ABB RobotStudio station: CubesMovement_20241125-112948.rsstn

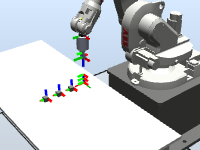
Station CubesMovement (saved by RobotStudio 6.8.8307.1040)
Controller System1, task T_ROB1: task frame (RAPID world) sits at (0, 0, 520) mm in the station
Controller System1
  mechanical unit ROB_1: IRB1600_10_145__01, 6 joints, base frame (0, 0, 0) mm
Layout (positions relative to the parent item):
  - IRB1600_10_145__01 [mechanism, from Robots\IRB1600_10_145_G_01.rslib] at (0, 0, 520) mm; joint values [-0.0068, 0.3691, 0.5943, 0, 0.6074, 1.564] (rad or m)
  - base [part, from Desktop\подставка.rslib]
  - table [part, from Desktop\Стол сборка.rslib] at (677.65, -723.32, 0) mm, rotated rx 0 ry 0 rz 90 deg
  - toolGripper [mechanism, from Desktop\toolGripper.rslib] at (744.98, -5.05, 1101.68) mm, rotated rx 180 ry 0 rz 90 deg
  - cube_1 [part, from Desktop\cube.rslib] at (844.98, -5.05, 730.16) mm
  - cube_2 [part, from Desktop\cube.rslib] at (944.98, -5.05, 730.39) mm
  - cube_3 [part, from Desktop\cube.rslib] at (1044.98, -5.05, 730.61) mm
Attachment: wobjTable is attached to table
Attachment: toolGripper is attached to IRB1600_10_145__01 / Link6
Collision set CollisionSet_1: IRB1600_10_145__01, toolGripper, table against table, toolGripper, near miss 0 m
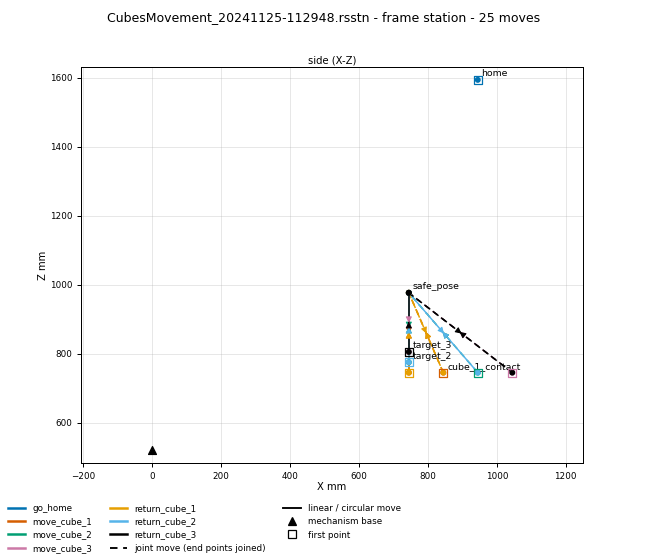
[picture p0: tool path of CubesMovement_20241125-112948.rsstn in frame station, 25 of 25 moves have a stored position in this frame; points joined in program order, loops and branches not executed]
Targets, tools, work objects and paths stored in the station, written as RAPID:
! task T_ROB1
MODULE CalibData
  PERS tooldata toolGripper:=[TRUE,[[0,0,160],[1,0,0,0]],[0.8,[0,0,1],[1,0,0,0],0,0,0]];
  TASK PERS wobjdata wobjTable:=[FALSE,TRUE,"",[[744.979,-5.048,210.071],[1,0,0,0]],[[0,0,0],[1,0,0,0]]];
ENDMODULE

! task T_ROB1
MODULE Module1
  CONST robtarget home:=[[944.855715851,0,1074],[0.5,0,0.866025404,0],[0,0,0,0],[9E+09,9E+09,9E+09,9E+09,9E+09,9E+09]];
  CONST robtarget cube_1_pose:=[[100,0,0],[1,0,0,0],[0,0,0,0],[9E+09,9E+09,9E+09,9E+09,9E+09,9E+09]];
  CONST robtarget cube_2_pose:=[[200,0,0],[1,0,0,0],[0,0,0,0],[9E+09,9E+09,9E+09,9E+09,9E+09,9E+09]];
  CONST robtarget cube_3_pose:=[[300,0,0],[1,0,0,0],[0,0,0,0],[9E+09,9E+09,9E+09,9E+09,9E+09,9E+09]];
  CONST robtarget tower_pose:=[[0,0,0],[1,0,0,0],[0,0,0,0],[9E+09,9E+09,9E+09,9E+09,9E+09,9E+09]];
  CONST robtarget cube_1_contact:=[[100,15,15],[0,0.707106781,0.707106781,0],[0,0,0,0],[9E+09,9E+09,9E+09,9E+09,9E+09,9E+09]];
  CONST robtarget cube_2_contact:=[[200,15,15],[0,0.707106781,0.707106781,0],[0,0,0,0],[9E+09,9E+09,9E+09,9E+09,9E+09,9E+09]];
  CONST robtarget cube_3_contact:=[[300,15,15],[0,0.707106781,0.707106781,0],[0,0,0,0],[9E+09,9E+09,9E+09,9E+09,9E+09,9E+09]];
  CONST robtarget target_1:=[[0,0,15],[0,0.707106781,0.707106781,0],[0,0,0,0],[9E+09,9E+09,9E+09,9E+09,9E+09,9E+09]];
  CONST robtarget target_2:=[[0,0,45],[0,0.707106781,0.707106781,0],[0,0,0,0],[9E+09,9E+09,9E+09,9E+09,9E+09,9E+09]];
  CONST robtarget target_3:=[[0,0,75],[0,0.707106781,0.707106781,0],[0,0,0,0],[9E+09,9E+09,9E+09,9E+09,9E+09,9E+09]];
  CONST robtarget safe_pose:=[[0.000003222,0.000000245,246.376418077],[0,0.707106781,0.707106781,0],[-1,-1,0,0],[9E+09,9E+09,9E+09,9E+09,9E+09,9E+09]];
  PROC go_home()
    MoveJ home,v100,fine,toolGripper\WObj:=wobj0;
  ENDPROC
  PROC main()
    go_home;
    move_cube_1;
    move_cube_2;
    move_cube_3;
    return_cube_3;
    return_cube_2;
    return_cube_1;
    go_home;
  ENDPROC
  PROC move_cube_1()
    MoveJ cube_1_contact,v100,fine,toolGripper\WObj:=wobjTable;
    PulseDO \High,do_GripClose;
    MoveJ safe_pose,v100,fine,toolGripper\WObj:=wobjTable;
    MoveL target_1,v100,fine,toolGripper\WObj:=wobjTable;
    PulseDO \High,do_GripOpen;
    MoveL safe_pose,v100,fine,toolGripper\WObj:=wobjTable;
  ENDPROC
  PROC move_cube_2()
    MoveJ cube_2_contact,v100,fine,toolGripper\WObj:=wobjTable;
    MoveJ safe_pose,v100,fine,toolGripper\WObj:=wobjTable;
    MoveL target_2,v100,fine,toolGripper\WObj:=wobjTable;
    MoveL safe_pose,v100,fine,toolGripper\WObj:=wobjTable;
  ENDPROC
  PROC move_cube_3()
    MoveJ cube_3_contact,v100,fine,toolGripper\WObj:=wobjTable;
    MoveJ safe_pose,v100,fine,toolGripper\WObj:=wobjTable;
    MoveL target_3,v100,fine,toolGripper\WObj:=wobjTable;
    MoveL safe_pose,v100,fine,toolGripper\WObj:=wobjTable;
  ENDPROC
  PROC return_cube_1()
    MoveL target_1,v100,fine,toolGripper\WObj:=wobjTable;
    MoveL safe_pose,v100,fine,toolGripper\WObj:=wobjTable;
    MoveJ cube_1_contact,v100,fine,toolGripper\WObj:=wobjTable;
    MoveJ safe_pose,v100,fine,toolGripper\WObj:=wobjTable;
  ENDPROC
  PROC return_cube_2()
    MoveL target_2,v100,fine,toolGripper\WObj:=wobjTable;
    MoveL safe_pose,v100,fine,toolGripper\WObj:=wobjTable;
    MoveJ cube_2_contact,v100,fine,toolGripper\WObj:=wobjTable;
    MoveJ safe_pose,v100,fine,toolGripper\WObj:=wobjTable;
  ENDPROC
  PROC return_cube_3()
    MoveL target_3,v100,fine,toolGripper\WObj:=wobjTable;
    MoveL safe_pose,v100,fine,toolGripper\WObj:=wobjTable;
    MoveJ cube_3_contact,v100,fine,toolGripper\WObj:=wobjTable;
    MoveJ safe_pose,v100,fine,toolGripper\WObj:=wobjTable;
  ENDPROC
ENDMODULE

